(* CODESYS project Tanque Industrial.project

Project tree, tasks and I/O mapping:
  Device : CODESYS Control Win V3, 3S - Smart Software Solutions GmbH, order no. 305021, version 3.5.11.30
    application Application
      libraries: Standard, * (System)
      task MainTask (cyclic, interval t#20ms, priority 1) calls PLC_PRG
      program PLC_PRG [LD]
      Symbols
*)

// Device/Application/PLC_PRG
PROGRAM PLC_PRG
VAR
	Encher:BOOL;
	Descarga:BOOL;
	Enchendo:BOOL;
	Esvaziando:BOOL;
	Valvula_Encher:BOOL;
	Valvula_Descarga:BOOL;
	Tempo_Encher:INT;
	Tempo_Esvaziar:INT; 
	tempo1_int:INT;
	tempo2_int:INT;	
	tempo_aux1:INT; 
	
	TOF_0: TOF;
	tempo1: TIME;
	TOF_1: TOF;
	tempo2: TIME;
	
	
END_VAR

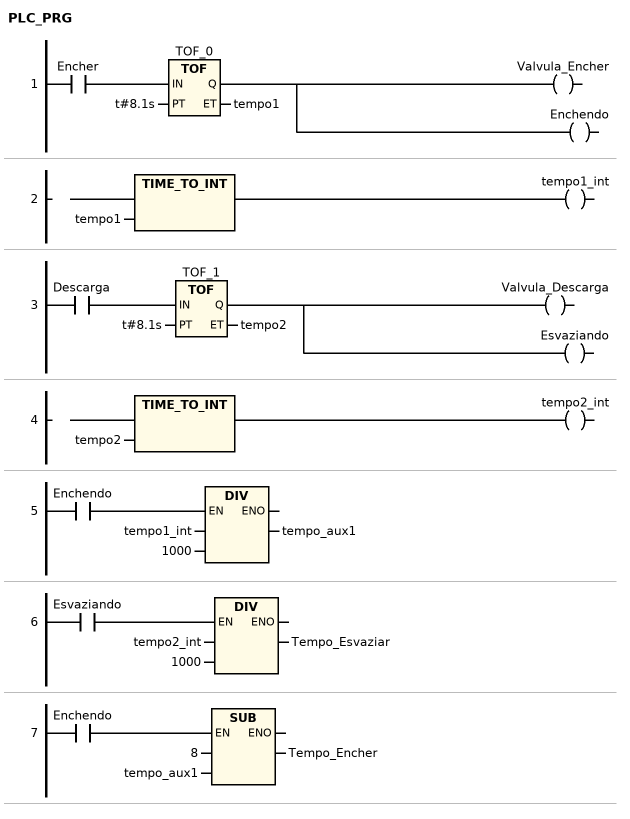
// NETWORK 1
TOF_0(IN := Encher, PT := t#8.1s, ET => tempo1); // TOF
Valvula_Encher := TOF_0.Q;
Enchendo := TOF_0.Q;

// NETWORK 2
tempo1_int := TIME_TO_INT(tempo1);

// NETWORK 3
TOF_1(IN := Descarga, PT := t#8.1s, ET => tempo2); // TOF
Valvula_Descarga := TOF_1.Q;
Esvaziando := TOF_1.Q;

// NETWORK 4
tempo2_int := TIME_TO_INT(tempo2);

// NETWORK 5
IF Enchendo THEN tempo_aux1 := tempo1_int / 1000; END_IF

// NETWORK 6
IF Esvaziando THEN Tempo_Esvaziar := tempo2_int / 1000; END_IF

// NETWORK 7
IF Enchendo THEN Tempo_Encher := 8 - tempo_aux1; END_IF

END_PROGRAM
